// TIA Portal V17 program export: 1 tag tables, 0 data types, 0 data blocks, 1 code blocks (in call order from the OBs), 2 instance data blocks

VAR_GLOBAL   // PLC tag table "Default tag table"
   Tag_1 AT %M1.0 : Bool;
   Tag_2 AT %M2.0 : Bool;
   Tag_3 AT %M3.0 : Bool;
   Tag_4 AT %M10.0 : Bool;
   Tag_5 AT %M20.0 : Bool;
END_VAR

ORGANIZATION_BLOCK "Main"   // OB1, LAD, ProgramCycle
TITLE = "Main Program Sweep (Cycle)"
{ S7_Optimized_Access := 'TRUE' }
VERSION : 0.1
// stored: AutoNumber true, IsIECCheckEnabled false, SetENOAutomatically false
   VAR_INPUT
      Initial_Call : Bool;   // Initial call of this OB
      Remanence : Bool;   // =True, if remanent data are available
   END_VAR
   VAR_TEMP   // added for the SCL form of the ladder/FBD networks
      _w1 : Bool;
   END_VAR
BEGIN

REGION Network 1
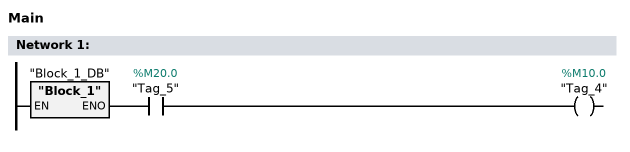
   RUNG wire#powerrail
      "Block_1_DB"()
      Contact( "Tag_5" )
      Coil( "Tag_4" )
   END_RUNG
   // the same network as SCL:
   "Block_1_DB"(ENO => #_w1);   // "Block_1"
   "Tag_4" := #_w1 AND "Tag_5";
END_REGION
END_ORGANIZATION_BLOCK

DATA_BLOCK "Block_1_DB"   // DB2
VERSION : 0.1
// stored: AutoNumber true, InstanceOfName Block_1, InstanceOfType FB
"Block_1"
BEGIN
END_DATA_BLOCK

DATA_BLOCK "Block_2_DB"   // DB1
VERSION : 0.1
// stored: AutoNumber true, InstanceOfName Block_2, InstanceOfType FB
"Block_2"
   // VAR_INPUT
   //    "1" : Bool;
   // END_VAR
   // VAR_OUTPUT
   //    "2" : Bool;
   // END_VAR
BEGIN
END_DATA_BLOCK
